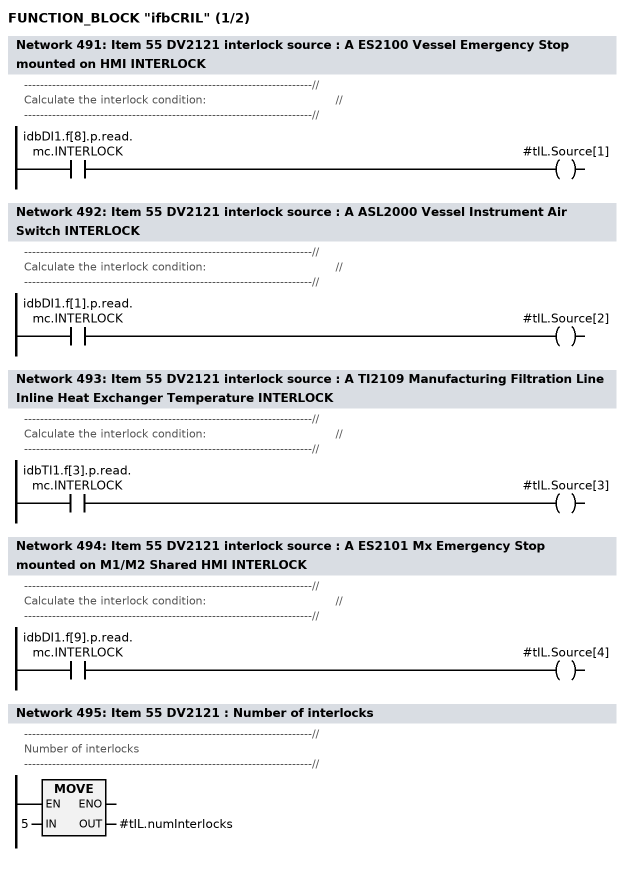
    A idbDI1.f[8].p.read.mc.INTERLOCK;
    = #tIL.Source[1];

NETWORK
TITLE = Item 55 DV2121 interlock source : A ASL2000 Vessel Instrument Air Switch INTERLOCK
    //------------------------------------------------------------------------//
    // Calculate the interlock condition:                                     //
    //------------------------------------------------------------------------//
    A idbDI1.f[1].p.read.mc.INTERLOCK;
    = #tIL.Source[2];

NETWORK
TITLE = Item 55 DV2121 interlock source : A TI2109 Manufacturing Filtration Line Inline Heat Exchanger Temperature INTERLOCK
    //------------------------------------------------------------------------//
    // Calculate the interlock condition:                                     //
    //------------------------------------------------------------------------//
    A idbTI1.f[3].p.read.mc.INTERLOCK;
    = #tIL.Source[3];

NETWORK
TITLE = Item 55 DV2121 interlock source : A ES2101 Mx Emergency Stop mounted on M1/M2 Shared HMI INTERLOCK
    //------------------------------------------------------------------------//
    // Calculate the interlock condition:                                     //
    //------------------------------------------------------------------------//
    A idbDI1.f[9].p.read.mc.INTERLOCK;
    = #tIL.Source[4];


NETWORK
TITLE = Item 55 DV2121 : Number of interlocks
    //------------------------------------------------------------------------//
    // Number of interlocks
    //------------------------------------------------------------------------//
    L 5;
    T #tIL.numInterlocks;

NETWORK
TITLE = Item 55 DV2121 : Aggregate individual interlocks into overall INTERLOCK flag
    //------------------------------------------------------------------------//
    // Determine if an interlock is raised:                                   //
    //------------------------------------------------------------------------//
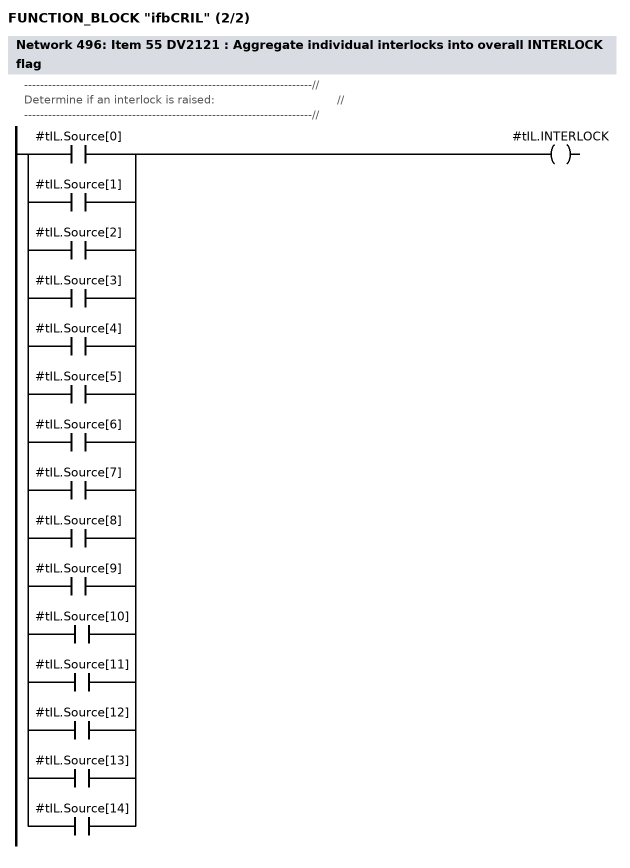
    O #tIL.Source[0];
    O #tIL.Source[1];
    O #tIL.Source[2];
    O #tIL.Source[3];
    O #tIL.Source[4];
    O #tIL.Source[5];
    O #tIL.Source[6];
    O #tIL.Source[7];
    O #tIL.Source[8];
    O #tIL.Source[9];
    O #tIL.Source[10];
    O #tIL.Source[11];
    O #tIL.Source[12];
    O #tIL.Source[13];
    O #tIL.Source[14];
    = #tIL.INTERLOCK;

NETWORK
TITLE = Item 55 DV2121 : Update the instance data
    //------------------------------------------------------------------------//
    // Update the instance DB with the calculated interlock flags:            //
    //------------------------------------------------------------------------//
    CALL MOVE
    {value_type := 'Variant'}
    (   IN                   := #tIL ,
        OUT                  := #p[55]
    );

NETWORK
TITLE = Item 56 DV2135 : SMFLx filter outlet drain valve initialise variables
    //------------------------------------------------------------------------//
    // CRITICAL INTERLOCK   CRITICAL INTERLOCK   CRITICAL INTERLOCK   CRITICA //
    // CRITICAL INTERLOCK   CRITICAL INTERLOCK   CRITICAL INTERLOCK   CRITICA //
    //                                                                        //
    // Clear the interlock flag:                                              //
    //------------------------------------------------------------------------//
    A "alwaysLow";
    = #tIL.INTERLOCK;

    //------------------------------------------------------------------------//
    // Clear all interlock values to initialise them to off:                  //
    //------------------------------------------------------------------------//
    CALL FILL_BLK
    {value_type := 'Bool', count_type := 'UInt'}
    (   IN                   := 0 ,
        COUNT                := 15 ,
        OUT                  := #tIL.Source[0]
    );


NETWORK
TITLE = Item 56 DV2135 interlock source : AN ZSC2111 MMFLx Filtration Inlet Flowpath Indicator IN   AN ZSC2109 SMFLx Filtration Line outlet Flowpath Indicator IN
    //------------------------------------------------------------------------//
    // Calculate the interlock condition:                                     //
    //------------------------------------------------------------------------//
    AN(;
    L "idbZSC2".f[11].p.read.mc.STATE;
    L "dbCONST".BLK.ZSC2.STATE.IN;
    ==I;
    );
AN(;
    L "idbZSC2".f[10].p.read.mc.STATE;
    L "dbCONST".BLK.ZSC2.STATE.IN;
    ==I;
    );
    = #tIL.Source[0];

NETWORK
TITLE = Item 56 DV2135 interlock source : A RD2101 Vessel Burst Disc ALARM
    //------------------------------------------------------------------------//
    // Calculate the interlock condition:                                     //
    //------------------------------------------------------------------------//
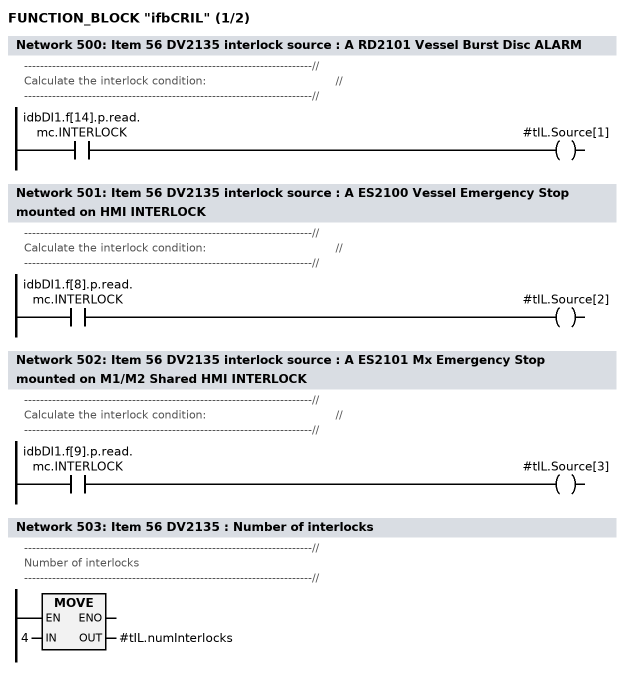
    A idbDI1.f[14].p.read.mc.INTERLOCK;
    = #tIL.Source[1];

NETWORK
TITLE = Item 56 DV2135 interlock source : A ES2100 Vessel Emergency Stop mounted on HMI INTERLOCK
    //------------------------------------------------------------------------//
    // Calculate the interlock condition:                                     //
    //------------------------------------------------------------------------//
    A idbDI1.f[8].p.read.mc.INTERLOCK;
    = #tIL.Source[2];

NETWORK
TITLE = Item 56 DV2135 interlock source : A ES2101 Mx Emergency Stop mounted on M1/M2 Shared HMI INTERLOCK
    //------------------------------------------------------------------------//
    // Calculate the interlock condition:                                     //
    //------------------------------------------------------------------------//
    A idbDI1.f[9].p.read.mc.INTERLOCK;
    = #tIL.Source[3];


NETWORK
TITLE = Item 56 DV2135 : Number of interlocks
    //------------------------------------------------------------------------//
    // Number of interlocks
    //------------------------------------------------------------------------//
    L 4;
    T #tIL.numInterlocks;

NETWORK
TITLE = Item 56 DV2135 : Aggregate individual interlocks into overall INTERLOCK flag
    //------------------------------------------------------------------------//
    // Determine if an interlock is raised:                                   //
    //------------------------------------------------------------------------//
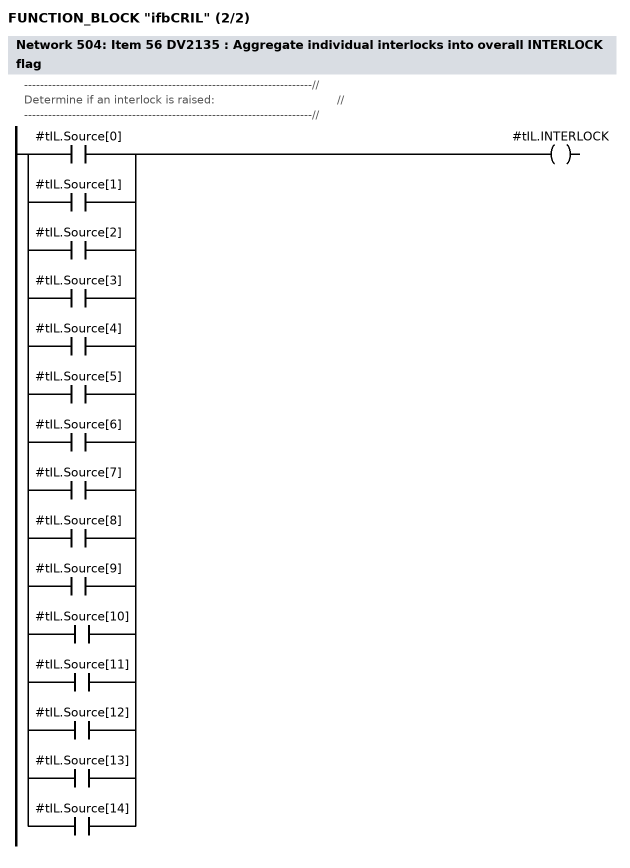
    O #tIL.Source[0];
    O #tIL.Source[1];
    O #tIL.Source[2];
    O #tIL.Source[3];
    O #tIL.Source[4];
    O #tIL.Source[5];
    O #tIL.Source[6];
    O #tIL.Source[7];
    O #tIL.Source[8];
    O #tIL.Source[9];
    O #tIL.Source[10];
    O #tIL.Source[11];
    O #tIL.Source[12];
    O #tIL.Source[13];
    O #tIL.Source[14];
    = #tIL.INTERLOCK;

NETWORK
TITLE = Item 56 DV2135 : Update the instance data
    //------------------------------------------------------------------------//
    // Update the instance DB with the calculated interlock flags:            //
    //------------------------------------------------------------------------//
    CALL MOVE
    {value_type := 'Variant'}
    (   IN                   := #tIL ,
        OUT                  := #p[56]
    );

NETWORK
TITLE = Item 57 DV2137 : SMFLx filter outlet valve initialise variables
    //------------------------------------------------------------------------//
    // CRITICAL INTERLOCK   CRITICAL INTERLOCK   CRITICAL INTERLOCK   CRITICA //
    // CRITICAL INTERLOCK   CRITICAL INTERLOCK   CRITICAL INTERLOCK   CRITICA //
    //                                                                        //
    // Clear the interlock flag:                                              //
    //------------------------------------------------------------------------//
    A "alwaysLow";
    = #tIL.INTERLOCK;

    //------------------------------------------------------------------------//
    // Clear all interlock values to initialise them to off:                  //
    //------------------------------------------------------------------------//
    CALL FILL_BLK
    {value_type := 'Bool', count_type := 'UInt'}
    (   IN                   := 0 ,
        COUNT                := 15 ,
        OUT                  := #tIL.Source[0]
    );


NETWORK
TITLE = Item 57 DV2137 interlock source : AN ZSC2111 MMFLx Filtration Inlet Flowpath Indicator IN   AN ZSC2109 SMFLx Filtration Line outlet Flowpath Indicator IN
    //------------------------------------------------------------------------//
    // Calculate the interlock condition:                                     //
    //------------------------------------------------------------------------//
    AN(;
    L "idbZSC2".f[11].p.read.mc.STATE;
    L "dbCONST".BLK.ZSC2.STATE.IN;
    ==I;
    );
AN(;
    L "idbZSC2".f[10].p.read.mc.STATE;
    L "dbCONST".BLK.ZSC2.STATE.IN;
    ==I;
    );
    = #tIL.Source[0];

NETWORK
TITLE = Item 57 DV2137 interlock source : A RD2101 Vessel Burst Disc ALARM
    //------------------------------------------------------------------------//
    // Calculate the interlock condition:                                     //
    //------------------------------------------------------------------------//
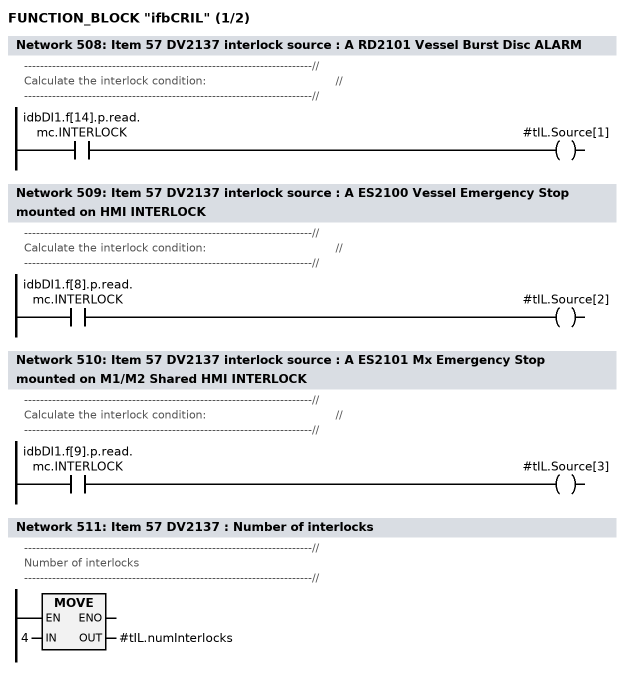
    A idbDI1.f[14].p.read.mc.INTERLOCK;
    = #tIL.Source[1];

NETWORK
TITLE = Item 57 DV2137 interlock source : A ES2100 Vessel Emergency Stop mounted on HMI INTERLOCK
    //------------------------------------------------------------------------//
    // Calculate the interlock condition:                                     //
    //------------------------------------------------------------------------//
    A idbDI1.f[8].p.read.mc.INTERLOCK;
    = #tIL.Source[2];

NETWORK
TITLE = Item 57 DV2137 interlock source : A ES2101 Mx Emergency Stop mounted on M1/M2 Shared HMI INTERLOCK
    //------------------------------------------------------------------------//
    // Calculate the interlock condition:                                     //
    //------------------------------------------------------------------------//
    A idbDI1.f[9].p.read.mc.INTERLOCK;
    = #tIL.Source[3];


NETWORK
TITLE = Item 57 DV2137 : Number of interlocks
    //------------------------------------------------------------------------//
    // Number of interlocks
    //------------------------------------------------------------------------//
    L 4;
    T #tIL.numInterlocks;

NETWORK
TITLE = Item 57 DV2137 : Aggregate individual interlocks into overall INTERLOCK flag
    //------------------------------------------------------------------------//
    // Determine if an interlock is raised:                                   //
    //------------------------------------------------------------------------//
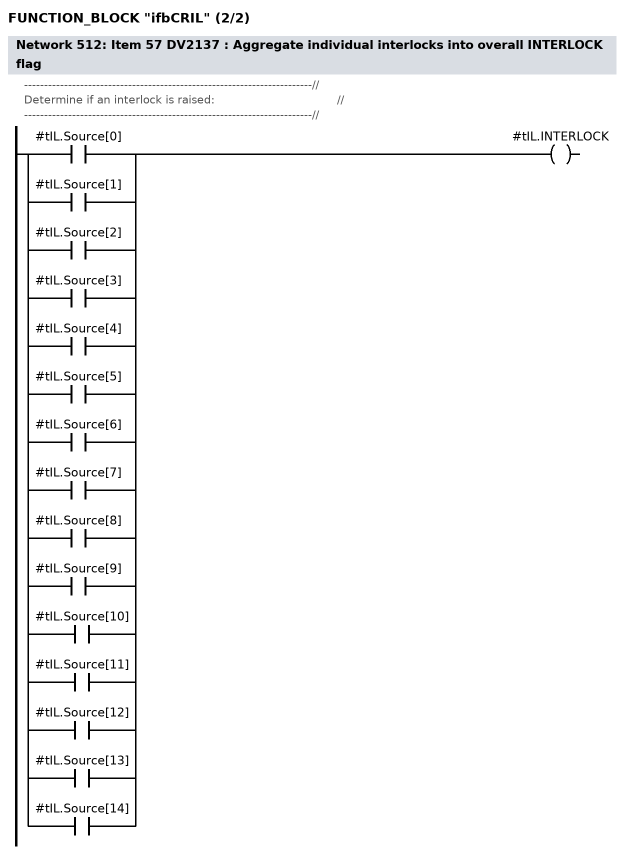
    O #tIL.Source[0];
    O #tIL.Source[1];
    O #tIL.Source[2];
    O #tIL.Source[3];
    O #tIL.Source[4];
    O #tIL.Source[5];
    O #tIL.Source[6];
    O #tIL.Source[7];
    O #tIL.Source[8];
    O #tIL.Source[9];
    O #tIL.Source[10];
    O #tIL.Source[11];
    O #tIL.Source[12];
    O #tIL.Source[13];
    O #tIL.Source[14];
    = #tIL.INTERLOCK;

NETWORK
TITLE = Item 57 DV2137 : Update the instance data
    //------------------------------------------------------------------------//
    // Update the instance DB with the calculated interlock flags:            //
    //------------------------------------------------------------------------//
    CALL MOVE
    {value_type := 'Variant'}
    (   IN                   := #tIL ,
        OUT                  := #p[57]
    );

NETWORK
TITLE = Item 58 DV2171 : MMFLx filter inlet drain valve initialise variables
    //------------------------------------------------------------------------//
    // CRITICAL INTERLOCK   CRITICAL INTERLOCK   CRITICAL INTERLOCK   CRITICA //
    // CRITICAL INTERLOCK   CRITICAL INTERLOCK   CRITICAL INTERLOCK   CRITICA //
    //                                                                        //
    // Clear the interlock flag:                                              //
    //------------------------------------------------------------------------//
    A "alwaysLow";
    = #tIL.INTERLOCK;

    //------------------------------------------------------------------------//
    // Clear all interlock values to initialise them to off:                  //
    //------------------------------------------------------------------------//
    CALL FILL_BLK
    {value_type := 'Bool', count_type := 'UInt'}
    (   IN                   := 0 ,
        COUNT                := 15 ,
        OUT                  := #tIL.Source[0]
    );


NETWORK
TITLE = Item 58 DV2171 interlock source : AN ZSC2113 MMFLx Filtration Inlet Flowpath Indicator IN   AN ZSC2115 MMFLx Filtration Inlet CIP & SIP Flowpath Indicator IN
    //------------------------------------------------------------------------//
    // Calculate the interlock condition:                                     //
    //------------------------------------------------------------------------//
    AN(;
    L "idbZSC2".f[12].p.read.mc.STATE;
    L "dbCONST".BLK.ZSC2.STATE.IN;
    ==I;
    );
AN(;
    L "idbZSC2".f[13].p.read.mc.STATE;
    L "dbCONST".BLK.ZSC2.STATE.IN;
    ==I;
    );
    = #tIL.Source[0];

NETWORK
TITLE = Item 58 DV2171 interlock source : AN ZSC2115 MMFLx Filtration Inlet CIP & SIP Flowpath Indicator IN
    //------------------------------------------------------------------------//
    // Calculate the interlock condition:                                     //
    //------------------------------------------------------------------------//
    AN(;
    L "idbZSC2".f[13].p.read.mc.STATE;
    L "dbCONST".BLK.ZSC2.STATE.IN;
    ==I;
    );
    = #tIL.Source[1];

NETWORK
TITLE = Item 58 DV2171 interlock source : A RD2101 Vessel Burst Disc ALARM
    //------------------------------------------------------------------------//
    // Calculate the interlock condition:                                     //
    //------------------------------------------------------------------------//
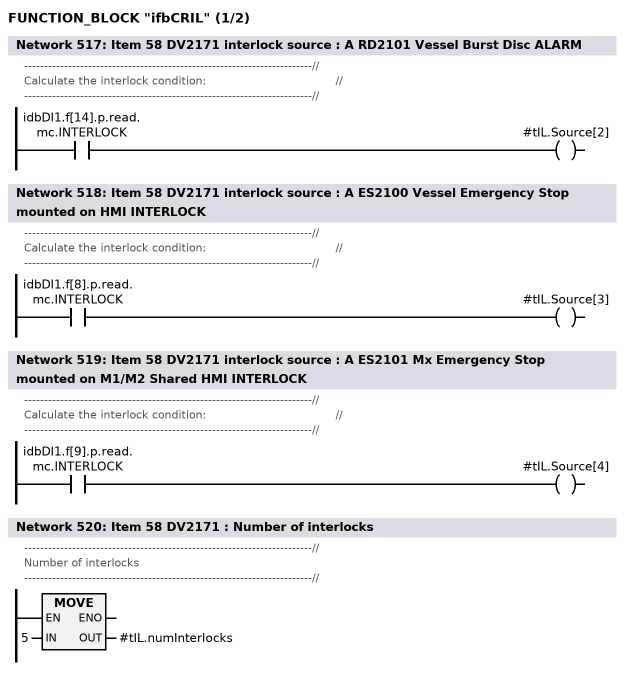
    A idbDI1.f[14].p.read.mc.INTERLOCK;
    = #tIL.Source[2];

NETWORK
TITLE = Item 58 DV2171 interlock source : A ES2100 Vessel Emergency Stop mounted on HMI INTERLOCK
    //------------------------------------------------------------------------//
    // Calculate the interlock condition:                                     //
    //------------------------------------------------------------------------//
    A idbDI1.f[8].p.read.mc.INTERLOCK;
    = #tIL.Source[3];

NETWORK
TITLE = Item 58 DV2171 interlock source : A ES2101 Mx Emergency Stop mounted on M1/M2 Shared HMI INTERLOCK
    //------------------------------------------------------------------------//
    // Calculate the interlock condition:                                     //
    //------------------------------------------------------------------------//
    A idbDI1.f[9].p.read.mc.INTERLOCK;
    = #tIL.Source[4];


NETWORK
TITLE = Item 58 DV2171 : Number of interlocks
    //------------------------------------------------------------------------//
    // Number of interlocks
    //------------------------------------------------------------------------//
    L 5;
    T #tIL.numInterlocks;

NETWORK
TITLE = Item 58 DV2171 : Aggregate individual interlocks into overall INTERLOCK flag
    //------------------------------------------------------------------------//
    // Determine if an interlock is raised:                                   //
    //------------------------------------------------------------------------//
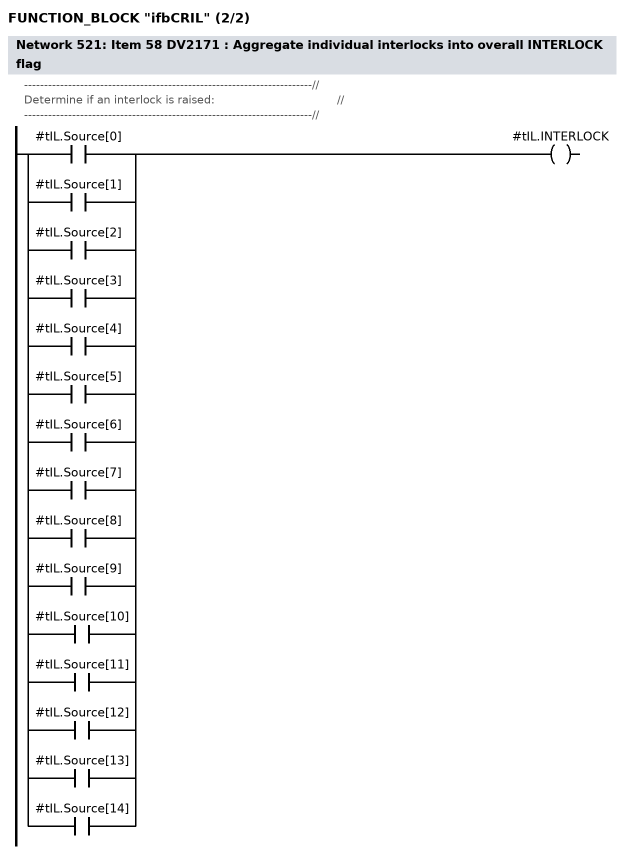
    O #tIL.Source[0];
    O #tIL.Source[1];
    O #tIL.Source[2];
    O #tIL.Source[3];
    O #tIL.Source[4];
    O #tIL.Source[5];
    O #tIL.Source[6];
    O #tIL.Source[7];
    O #tIL.Source[8];
    O #tIL.Source[9];
    O #tIL.Source[10];
    O #tIL.Source[11];
    O #tIL.Source[12];
    O #tIL.Source[13];
    O #tIL.Source[14];
    = #tIL.INTERLOCK;

NETWORK
TITLE = Item 58 DV2171 : Update the instance data
    //------------------------------------------------------------------------//
    // Update the instance DB with the calculated interlock flags:            //
    //------------------------------------------------------------------------//
    CALL MOVE
    {value_type := 'Variant'}
    (   IN                   := #tIL ,
        OUT                  := #p[58]
    );

NETWORK
TITLE = Item 59 DV2173 : MMFLx Inline Heat Exchanger inlet valve initialise variables
    //------------------------------------------------------------------------//
    // CRITICAL INTERLOCK   CRITICAL INTERLOCK   CRITICAL INTERLOCK   CRITICA //
    // CRITICAL INTERLOCK   CRITICAL INTERLOCK   CRITICAL INTERLOCK   CRITICA //
    //                                                                        //
    // Clear the interlock flag:                                              //
    //------------------------------------------------------------------------//
    A "alwaysLow";
    = #tIL.INTERLOCK;

    //------------------------------------------------------------------------//
    // Clear all interlock values to initialise them to off:                  //
    //------------------------------------------------------------------------//
    CALL FILL_BLK
    {value_type := 'Bool', count_type := 'UInt'}
    (   IN                   := 0 ,
        COUNT                := 15 ,
        OUT                  := #tIL.Source[0]
    );


NETWORK
TITLE = Item 59 DV2173 interlock source : AN ZSC2113 MMFLx Filtration Inlet Flowpath Indicator IN   AN ZSC2115 MMFLx Filtration Inlet CIP & SIP Flowpath Indicator IN
    //------------------------------------------------------------------------//
    // Calculate the interlock condition:                                     //
    //------------------------------------------------------------------------//
    AN(;
    L "idbZSC2".f[12].p.read.mc.STATE;
    L "dbCONST".BLK.ZSC2.STATE.IN;
    ==I;
    );
AN(;
    L "idbZSC2".f[13].p.read.mc.STATE;
    L "dbCONST".BLK.ZSC2.STATE.IN;
    ==I;
    );
    = #tIL.Source[0];

NETWORK
TITLE = Item 59 DV2173 interlock source : A RD2101 Vessel Burst Disc ALARM
    //------------------------------------------------------------------------//
    // Calculate the interlock condition:                                     //
    //------------------------------------------------------------------------//
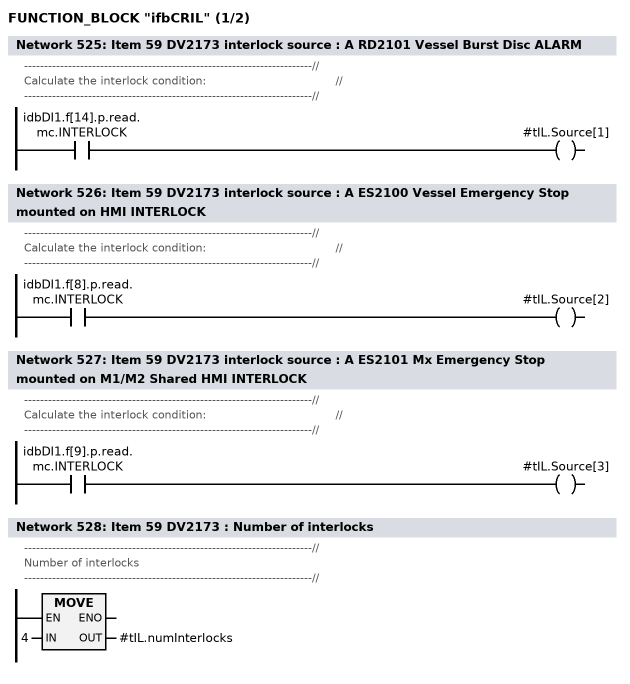
    A idbDI1.f[14].p.read.mc.INTERLOCK;
    = #tIL.Source[1];

NETWORK
TITLE = Item 59 DV2173 interlock source : A ES2100 Vessel Emergency Stop mounted on HMI INTERLOCK
    //------------------------------------------------------------------------//
    // Calculate the interlock condition:                                     //
    //------------------------------------------------------------------------//
    A idbDI1.f[8].p.read.mc.INTERLOCK;
    = #tIL.Source[2];

NETWORK
TITLE = Item 59 DV2173 interlock source : A ES2101 Mx Emergency Stop mounted on M1/M2 Shared HMI INTERLOCK
    //------------------------------------------------------------------------//
    // Calculate the interlock condition:                                     //
    //------------------------------------------------------------------------//
    A idbDI1.f[9].p.read.mc.INTERLOCK;
    = #tIL.Source[3];


NETWORK
TITLE = Item 59 DV2173 : Number of interlocks
    //------------------------------------------------------------------------//
    // Number of interlocks
    //------------------------------------------------------------------------//
    L 4;
    T #tIL.numInterlocks;

NETWORK
TITLE = Item 59 DV2173 : Aggregate individual interlocks into overall INTERLOCK flag
    //------------------------------------------------------------------------//
    // Determine if an interlock is raised:                                   //
    //------------------------------------------------------------------------//
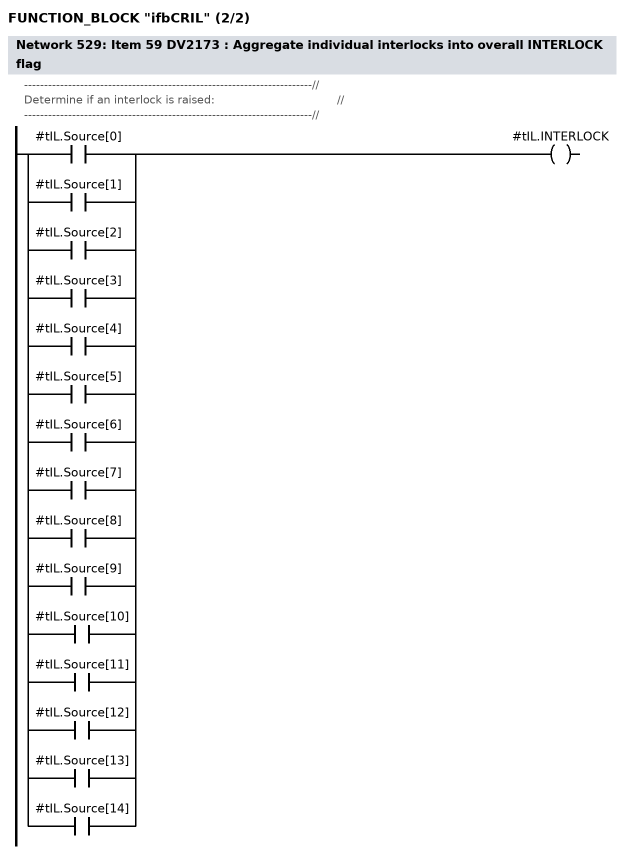
    O #tIL.Source[0];
    O #tIL.Source[1];
    O #tIL.Source[2];
    O #tIL.Source[3];
    O #tIL.Source[4];
    O #tIL.Source[5];
    O #tIL.Source[6];
    O #tIL.Source[7];
    O #tIL.Source[8];
    O #tIL.Source[9];
    O #tIL.Source[10];
    O #tIL.Source[11];
    O #tIL.Source[12];
    O #tIL.Source[13];
    O #tIL.Source[14];
    = #tIL.INTERLOCK;

NETWORK
TITLE = Item 59 DV2173 : Update the instance data
    //------------------------------------------------------------------------//
    // Update the instance DB with the calculated interlock flags:            //
    //------------------------------------------------------------------------//
    CALL MOVE
    {value_type := 'Variant'}
    (   IN                   := #tIL ,
        OUT                  := #p[59]
    );

NETWORK
TITLE = Item 60 DV3101 : Vent Valve initialise variables
    //------------------------------------------------------------------------//
    // CRITICAL INTERLOCK   CRITICAL INTERLOCK   CRITICAL INTERLOCK   CRITICA //
    // CRITICAL INTERLOCK   CRITICAL INTERLOCK   CRITICAL INTERLOCK   CRITICA //
    //                                                                        //
    // Clear the interlock flag:                                              //
    //------------------------------------------------------------------------//
    A "alwaysLow";
    = #tIL.INTERLOCK;

    //------------------------------------------------------------------------//
    // Clear all interlock values to initialise them to off:                  //
    //------------------------------------------------------------------------//
    CALL FILL_BLK
    {value_type := 'Bool', count_type := 'UInt'}
    (   IN                   := 0 ,
        COUNT                := 15 ,
        OUT                  := #tIL.Source[0]
    );


NETWORK
TITLE = Item 60 DV3101 interlock source : A RD3101 Vessel Burst Disc ALARM
    //------------------------------------------------------------------------//
    // Calculate the interlock condition:                                     //
    //------------------------------------------------------------------------//
    A idbDI1.f[15].p.read.mc.INTERLOCK;
    = #tIL.Source[0];

NETWORK
TITLE = Item 60 DV3101 interlock source : A ES3100 Vessel Emergency Stop mounted on HMI INTERLOCK
    //------------------------------------------------------------------------//
    // Calculate the interlock condition:                                     //
    //------------------------------------------------------------------------//
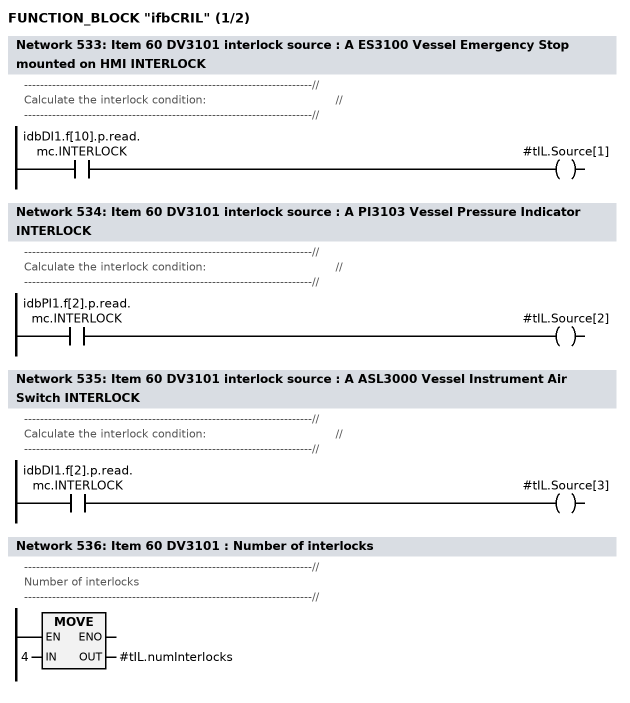
    A idbDI1.f[10].p.read.mc.INTERLOCK;
    = #tIL.Source[1];

NETWORK
TITLE = Item 60 DV3101 interlock source : A PI3103 Vessel Pressure Indicator INTERLOCK
    //------------------------------------------------------------------------//
    // Calculate the interlock condition:                                     //
    //------------------------------------------------------------------------//
    A idbPI1.f[2].p.read.mc.INTERLOCK;
    = #tIL.Source[2];

NETWORK
TITLE = Item 60 DV3101 interlock source : A ASL3000 Vessel Instrument Air Switch INTERLOCK
    //------------------------------------------------------------------------//
    // Calculate the interlock condition:                                     //
    //------------------------------------------------------------------------//
    A idbDI1.f[2].p.read.mc.INTERLOCK;
    = #tIL.Source[3];


NETWORK
TITLE = Item 60 DV3101 : Number of interlocks
    //------------------------------------------------------------------------//
    // Number of interlocks
    //------------------------------------------------------------------------//
    L 4;
    T #tIL.numInterlocks;

NETWORK
TITLE = Item 60 DV3101 : Aggregate individual interlocks into overall INTERLOCK flag
    //------------------------------------------------------------------------//
    // Determine if an interlock is raised:                                   //
    //------------------------------------------------------------------------//
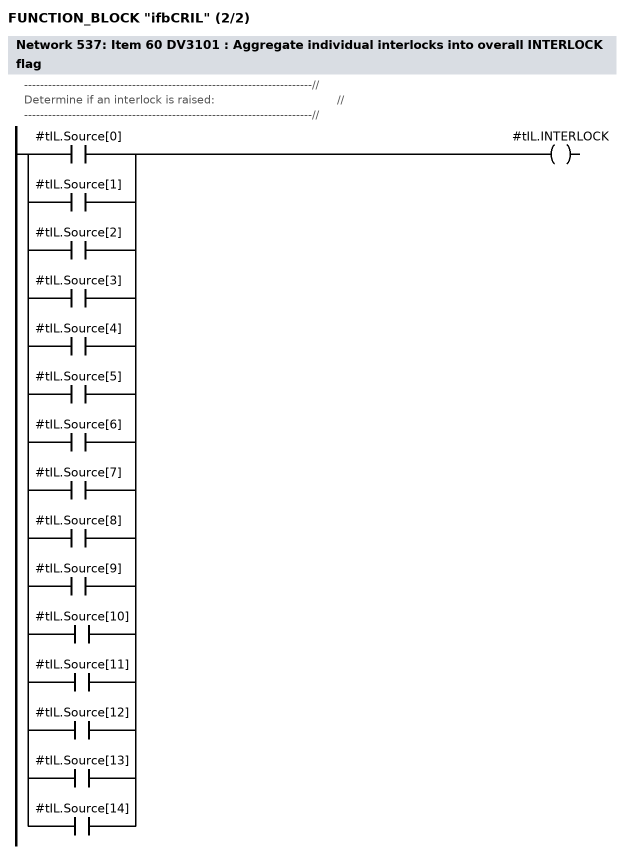
    O #tIL.Source[0];
    O #tIL.Source[1];
    O #tIL.Source[2];
    O #tIL.Source[3];
    O #tIL.Source[4];
    O #tIL.Source[5];
    O #tIL.Source[6];
    O #tIL.Source[7];
    O #tIL.Source[8];
    O #tIL.Source[9];
    O #tIL.Source[10];
    O #tIL.Source[11];
    O #tIL.Source[12];
    O #tIL.Source[13];
    O #tIL.Source[14];
    = #tIL.INTERLOCK;

NETWORK
TITLE = Item 60 DV3101 : Update the instance data
    //------------------------------------------------------------------------//
    // Update the instance DB with the calculated interlock flags:            //
    //------------------------------------------------------------------------//
    CALL MOVE
    {value_type := 'Variant'}
    (   IN                   := #tIL ,
        OUT                  := #p[60]
    );

NETWORK
TITLE = Item 61 DV3103 : HP CA Supply Valve initialise variables
    //------------------------------------------------------------------------//
    // CRITICAL INTERLOCK   CRITICAL INTERLOCK   CRITICAL INTERLOCK   CRITICA //
    // CRITICAL INTERLOCK   CRITICAL INTERLOCK   CRITICAL INTERLOCK   CRITICA //
    //                                                                        //
    // Clear the interlock flag:                                              //
    //------------------------------------------------------------------------//
    A "alwaysLow";
    = #tIL.INTERLOCK;

    //------------------------------------------------------------------------//
    // Clear all interlock values to initialise them to off:                  //
    //------------------------------------------------------------------------//
    CALL FILL_BLK
    {value_type := 'Bool', count_type := 'UInt'}
    (   IN                   := 0 ,
        COUNT                := 15 ,
        OUT                  := #tIL.Source[0]
    );


NETWORK
TITLE = Item 61 DV3103 interlock source : A RD3101 Vessel Burst Disc ALARM
    //------------------------------------------------------------------------//
    // Calculate the interlock condition:                                     //
    //------------------------------------------------------------------------//
    A idbDI1.f[15].p.read.mc.INTERLOCK;
    = #tIL.Source[0];

NETWORK
TITLE = Item 61 DV3103 interlock source : A ES3100 Vessel Emergency Stop mounted on HMI INTERLOCK
    //------------------------------------------------------------------------//
    // Calculate the interlock condition:                                     //
    //------------------------------------------------------------------------//
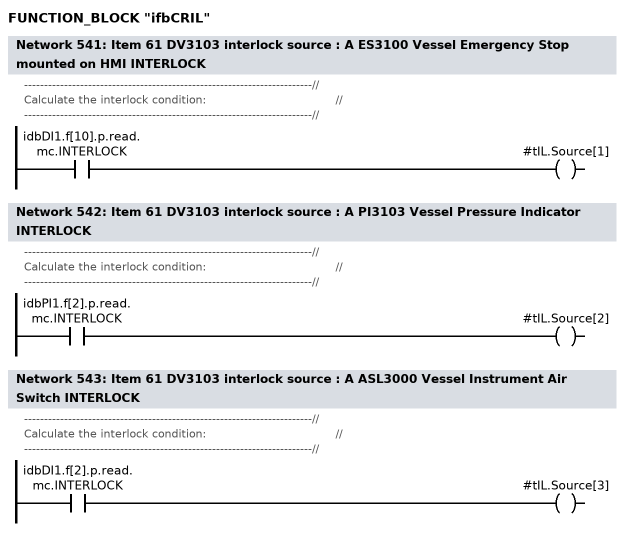
    A idbDI1.f[10].p.read.mc.INTERLOCK;
    = #tIL.Source[1];

NETWORK
TITLE = Item 61 DV3103 interlock source : A PI3103 Vessel Pressure Indicator INTERLOCK
    //------------------------------------------------------------------------//
    // Calculate the interlock condition:                                     //
    //------------------------------------------------------------------------//
    A idbPI1.f[2].p.read.mc.INTERLOCK;
    = #tIL.Source[2];

NETWORK
TITLE = Item 61 DV3103 interlock source : A ASL3000 Vessel Instrument Air Switch INTERLOCK
    //------------------------------------------------------------------------//
    // Calculate the interlock condition:                                     //
    //------------------------------------------------------------------------//
    A idbDI1.f[2].p.read.mc.INTERLOCK;
    = #tIL.Source[3];

NETWORK
TITLE = Item 61 DV3103 interlock source : AN ZSC3101 Vessel Manway Closed Indicator CLOSED
    //------------------------------------------------------------------------//
    // Calculate the interlock condition:                                     //
    //------------------------------------------------------------------------//
    AN(;
    L "idbZSC1".f[2].p.read.mc.STATE;
    L "dbCONST".BLK.ZSC1.STATE.CLOSED;
    ==I;
    );
    = #tIL.Source[4];


NETWORK
TITLE = Item 61 DV3103 : Number of interlocks
    //------------------------------------------------------------------------//
    // Number of interlocks
    //------------------------------------------------------------------------//
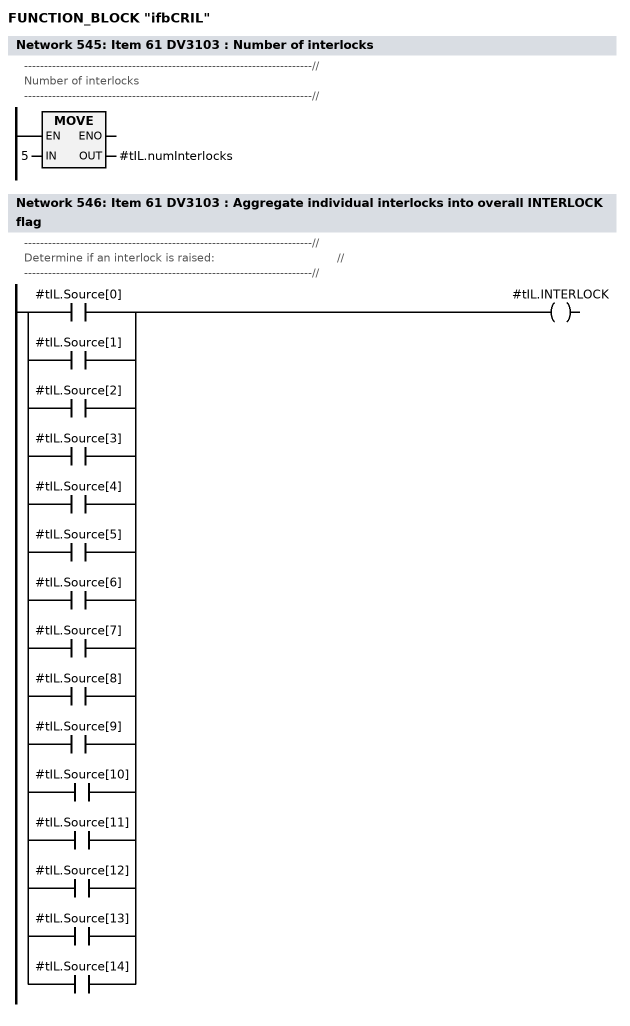
    L 5;
    T #tIL.numInterlocks;

NETWORK
TITLE = Item 61 DV3103 : Aggregate individual interlocks into overall INTERLOCK flag
    //------------------------------------------------------------------------//
    // Determine if an interlock is raised:                                   //
    //------------------------------------------------------------------------//
    O #tIL.Source[0];
    O #tIL.Source[1];
    O #tIL.Source[2];
    O #tIL.Source[3];
    O #tIL.Source[4];
    O #tIL.Source[5];
    O #tIL.Source[6];
    O #tIL.Source[7];
    O #tIL.Source[8];
    O #tIL.Source[9];
    O #tIL.Source[10];
    O #tIL.Source[11];
    O #tIL.Source[12];
    O #tIL.Source[13];
    O #tIL.Source[14];
    = #tIL.INTERLOCK;

NETWORK
TITLE = Item 61 DV3103 : Update the instance data
    //------------------------------------------------------------------------//
    // Update the instance DB with the calculated interlock flags:            //
    //------------------------------------------------------------------------//
    CALL MOVE
    {value_type := 'Variant'}
    (   IN                   := #tIL ,
        OUT                  := #p[61]
    );

NETWORK
TITLE = Item 62 DV3105 : LP CA Supply Valve initialise variables
    //------------------------------------------------------------------------//
    // CRITICAL INTERLOCK   CRITICAL INTERLOCK   CRITICAL INTERLOCK   CRITICA //
    // CRITICAL INTERLOCK   CRITICAL INTERLOCK   CRITICAL INTERLOCK   CRITICA //
    //                                                                        //
    // Clear the interlock flag:                                              //
    //------------------------------------------------------------------------//
    A "alwaysLow";
    = #tIL.INTERLOCK;

    //------------------------------------------------------------------------//
    // Clear all interlock values to initialise them to off:                  //
    //------------------------------------------------------------------------//
    CALL FILL_BLK
    {value_type := 'Bool', count_type := 'UInt'}
    (   IN                   := 0 ,
        COUNT                := 15 ,
        OUT                  := #tIL.Source[0]
    );


NETWORK
TITLE = Item 62 DV3105 interlock source : A RD3101 Vessel Burst Disc ALARM
    //------------------------------------------------------------------------//
    // Calculate the interlock condition:                                     //
    //------------------------------------------------------------------------//
    A idbDI1.f[15].p.read.mc.INTERLOCK;
    = #tIL.Source[0];

NETWORK
TITLE = Item 62 DV3105 interlock source : A ES3100 Vessel Emergency Stop mounted on HMI INTERLOCK
    //------------------------------------------------------------------------//
    // Calculate the interlock condition:                                     //
    //------------------------------------------------------------------------//
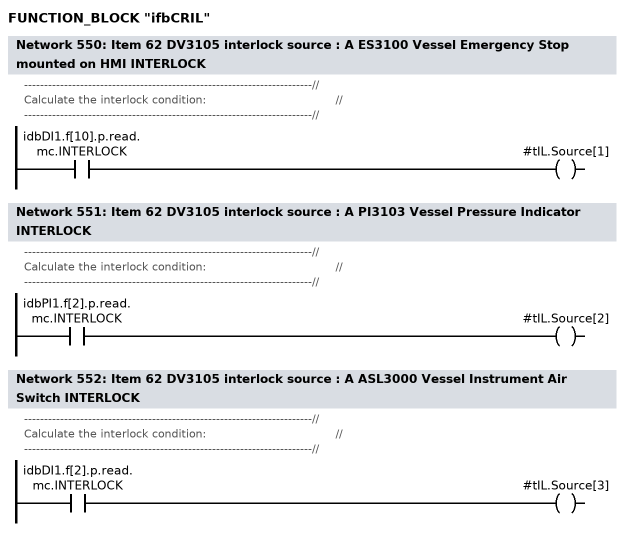
    A idbDI1.f[10].p.read.mc.INTERLOCK;
    = #tIL.Source[1];

NETWORK
TITLE = Item 62 DV3105 interlock source : A PI3103 Vessel Pressure Indicator INTERLOCK
    //------------------------------------------------------------------------//
    // Calculate the interlock condition:                                     //
    //------------------------------------------------------------------------//
    A idbPI1.f[2].p.read.mc.INTERLOCK;
    = #tIL.Source[2];

NETWORK
TITLE = Item 62 DV3105 interlock source : A ASL3000 Vessel Instrument Air Switch INTERLOCK
    //------------------------------------------------------------------------//
    // Calculate the interlock condition:                                     //
    //------------------------------------------------------------------------//
    A idbDI1.f[2].p.read.mc.INTERLOCK;
    = #tIL.Source[3];

NETWORK
TITLE = Item 62 DV3105 interlock source : AN ZSC3101 Vessel Manway Closed Indicator CLOSED
    //------------------------------------------------------------------------//
    // Calculate the interlock condition:                                     //
    //------------------------------------------------------------------------//
    AN(;
    L "idbZSC1".f[2].p.read.mc.STATE;
    L "dbCONST".BLK.ZSC1.STATE.CLOSED;
    ==I;
    );
    = #tIL.Source[4];


NETWORK
TITLE = Item 62 DV3105 : Number of interlocks
    //------------------------------------------------------------------------//
    // Number of interlocks
    //------------------------------------------------------------------------//
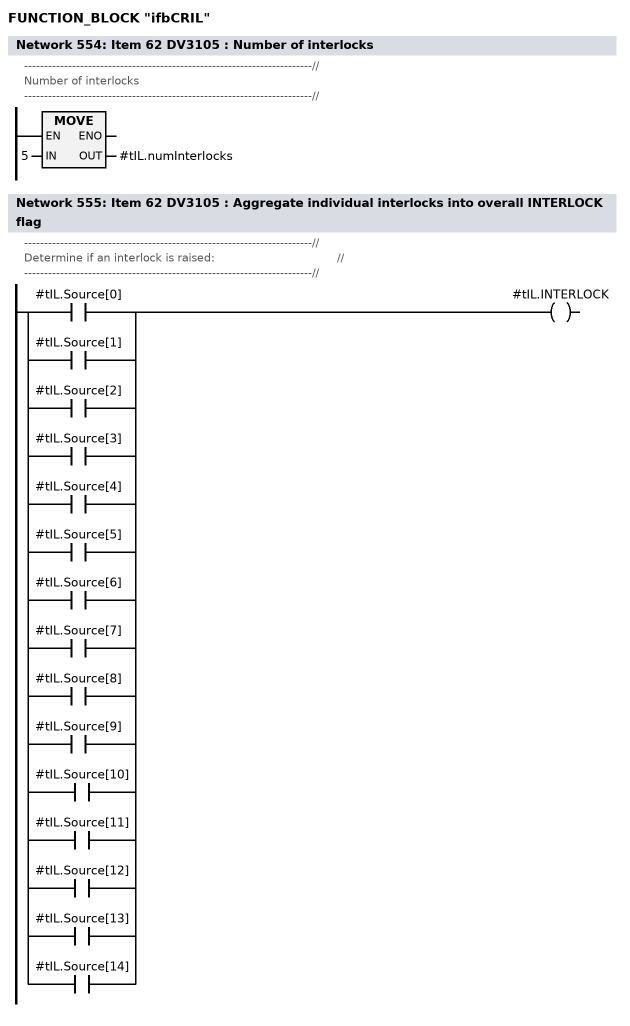
    L 5;
    T #tIL.numInterlocks;

NETWORK
TITLE = Item 62 DV3105 : Aggregate individual interlocks into overall INTERLOCK flag
    //------------------------------------------------------------------------//
    // Determine if an interlock is raised:                                   //
    //------------------------------------------------------------------------//
    O #tIL.Source[0];
    O #tIL.Source[1];
    O #tIL.Source[2];
    O #tIL.Source[3];
    O #tIL.Source[4];
    O #tIL.Source[5];
    O #tIL.Source[6];
    O #tIL.Source[7];
    O #tIL.Source[8];
    O #tIL.Source[9];
    O #tIL.Source[10];
    O #tIL.Source[11];
    O #tIL.Source[12];
    O #tIL.Source[13];
    O #tIL.Source[14];
    = #tIL.INTERLOCK;

NETWORK
TITLE = Item 62 DV3105 : Update the instance data
    //------------------------------------------------------------------------//
    // Update the instance DB with the calculated interlock flags:            //
    //------------------------------------------------------------------------//
    CALL MOVE
    {value_type := 'Variant'}
    (   IN                   := #tIL ,
        OUT                  := #p[62]
    );

NETWORK
TITLE = Item 63 DV3107 : Vacuum valve initialise variables
    //------------------------------------------------------------------------//
    // CRITICAL INTERLOCK   CRITICAL INTERLOCK   CRITICAL INTERLOCK   CRITICA //
    // CRITICAL INTERLOCK   CRITICAL INTERLOCK   CRITICAL INTERLOCK   CRITICA //
    //                                                                        //
    // Clear the interlock flag:                                              //
    //------------------------------------------------------------------------//
    A "alwaysLow";
    = #tIL.INTERLOCK;

    //------------------------------------------------------------------------//
    // Clear all interlock values to initialise them to off:                  //
    //------------------------------------------------------------------------//
    CALL FILL_BLK
    {value_type := 'Bool', count_type := 'UInt'}
    (   IN                   := 0 ,
        COUNT                := 15 ,
        OUT                  := #tIL.Source[0]
    );


NETWORK
TITLE = Item 63 DV3107 interlock source : A RD3101 Vessel Burst Disc ALARM
    //------------------------------------------------------------------------//
    // Calculate the interlock condition:                                     //
    //------------------------------------------------------------------------//
    A idbDI1.f[15].p.read.mc.INTERLOCK;
    = #tIL.Source[0];

NETWORK
TITLE = Item 63 DV3107 interlock source : A ES3100 Vessel Emergency Stop mounted on HMI INTERLOCK
    //------------------------------------------------------------------------//
    // Calculate the interlock condition:                                     //
    //------------------------------------------------------------------------//
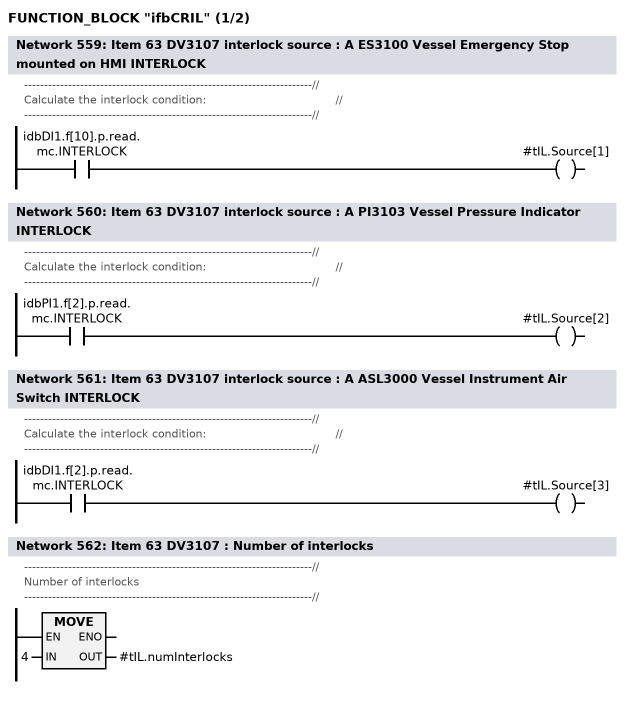
    A idbDI1.f[10].p.read.mc.INTERLOCK;
    = #tIL.Source[1];

NETWORK
TITLE = Item 63 DV3107 interlock source : A PI3103 Vessel Pressure Indicator INTERLOCK
    //------------------------------------------------------------------------//
    // Calculate the interlock condition:                                     //
    //------------------------------------------------------------------------//
    A idbPI1.f[2].p.read.mc.INTERLOCK;
    = #tIL.Source[2];

NETWORK
TITLE = Item 63 DV3107 interlock source : A ASL3000 Vessel Instrument Air Switch INTERLOCK
    //------------------------------------------------------------------------//
    // Calculate the interlock condition:                                     //
    //------------------------------------------------------------------------//
    A idbDI1.f[2].p.read.mc.INTERLOCK;
    = #tIL.Source[3];


NETWORK
TITLE = Item 63 DV3107 : Number of interlocks
    //------------------------------------------------------------------------//
    // Number of interlocks
    //------------------------------------------------------------------------//
    L 4;
    T #tIL.numInterlocks;

NETWORK
TITLE = Item 63 DV3107 : Aggregate individual interlocks into overall INTERLOCK flag
    //------------------------------------------------------------------------//
    // Determine if an interlock is raised:                                   //
    //------------------------------------------------------------------------//
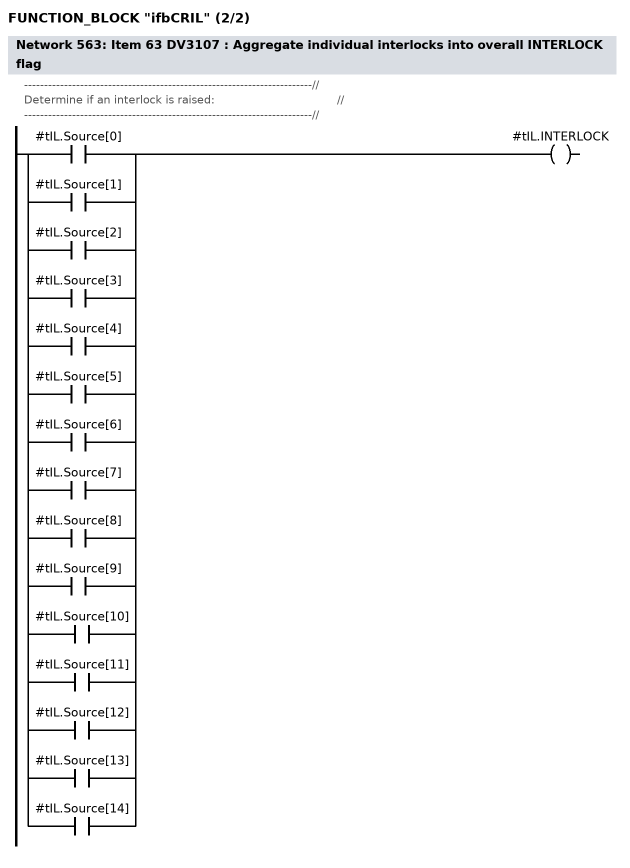
    O #tIL.Source[0];
    O #tIL.Source[1];
    O #tIL.Source[2];
    O #tIL.Source[3];
    O #tIL.Source[4];
    O #tIL.Source[5];
    O #tIL.Source[6];
    O #tIL.Source[7];
    O #tIL.Source[8];
    O #tIL.Source[9];
    O #tIL.Source[10];
    O #tIL.Source[11];
    O #tIL.Source[12];
    O #tIL.Source[13];
    O #tIL.Source[14];
    = #tIL.INTERLOCK;

NETWORK
TITLE = Item 63 DV3107 : Update the instance data
    //------------------------------------------------------------------------//
    // Update the instance DB with the calculated interlock flags:            //
    //------------------------------------------------------------------------//
    CALL MOVE
    {value_type := 'Variant'}
    (   IN                   := #tIL ,
        OUT                  := #p[63]
    );

NETWORK
TITLE = Item 64 DV3109 : PS Supply for WFI Loop initialise variables
    //------------------------------------------------------------------------//
    // CRITICAL INTERLOCK   CRITICAL INTERLOCK   CRITICAL INTERLOCK   CRITICA //
    // CRITICAL INTERLOCK   CRITICAL INTERLOCK   CRITICAL INTERLOCK   CRITICA //
    //                                                                        //
    // Clear the interlock flag:                                              //
    //------------------------------------------------------------------------//
    A "alwaysLow";
    = #tIL.INTERLOCK;

    //------------------------------------------------------------------------//
    // Clear all interlock values to initialise them to off:                  //
    //------------------------------------------------------------------------//
    CALL FILL_BLK
    {value_type := 'Bool', count_type := 'UInt'}
    (   IN                   := 0 ,
        COUNT                := 15 ,
        OUT                  := #tIL.Source[0]
    );


NETWORK
TITLE = Item 64 DV3109 interlock source : ON ZSC3107 Vessel inlet line Flowpath Indicator IN   ON ZSC3103 Vessel WFI Supply Flowpath Indicator IN
    //------------------------------------------------------------------------//
    // Calculate the interlock condition:                                     //
    //------------------------------------------------------------------------//
    ON(;
    L "idbZSC2".f[16].p.read.mc.STATE;
    L "dbCONST".BLK.ZSC2.STATE.IN;
    ==I;
    );
ON(;
    L "idbZSC2".f[14].p.read.mc.STATE;
    L "dbCONST".BLK.ZSC2.STATE.IN;
    ==I;
    );
    = #tIL.Source[0];

NETWORK
TITLE = Item 64 DV3109 interlock source : A DV3111 Vessel WFI Supply Valve OPENED
    //------------------------------------------------------------------------//
    // Calculate the interlock condition:                                     //
    //------------------------------------------------------------------------//
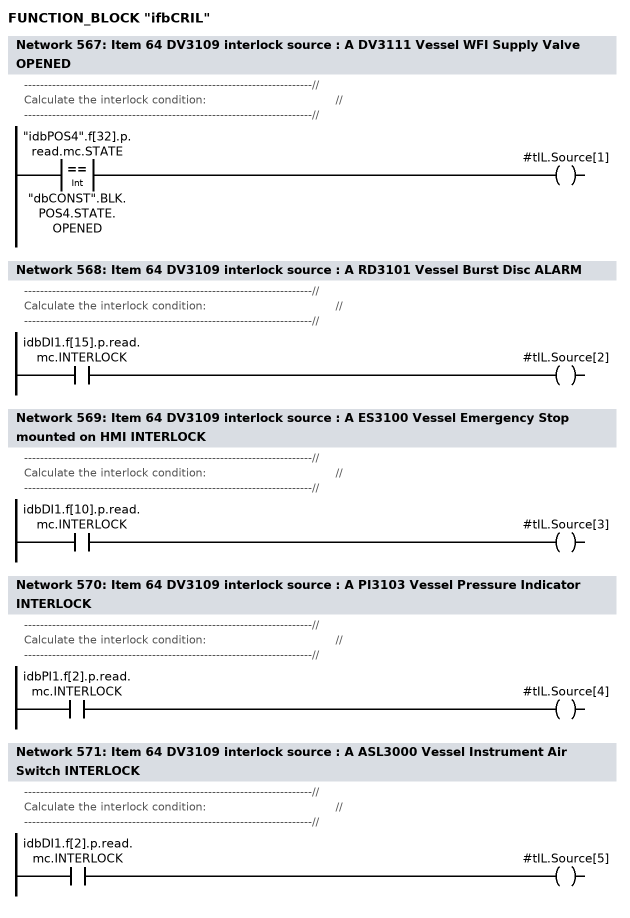
    A(;
    L "idbPOS4".f[32].p.read.mc.STATE;
    L "dbCONST".BLK.POS4.STATE.OPENED;
    ==I;
    );
    = #tIL.Source[1];

NETWORK
TITLE = Item 64 DV3109 interlock source : A RD3101 Vessel Burst Disc ALARM
    //------------------------------------------------------------------------//
    // Calculate the interlock condition:                                     //
    //------------------------------------------------------------------------//
    A idbDI1.f[15].p.read.mc.INTERLOCK;
    = #tIL.Source[2];

NETWORK
TITLE = Item 64 DV3109 interlock source : A ES3100 Vessel Emergency Stop mounted on HMI INTERLOCK
    //------------------------------------------------------------------------//
    // Calculate the interlock condition:                                     //
    //------------------------------------------------------------------------//
    A idbDI1.f[10].p.read.mc.INTERLOCK;
    = #tIL.Source[3];

NETWORK
TITLE = Item 64 DV3109 interlock source : A PI3103 Vessel Pressure Indicator INTERLOCK
    //------------------------------------------------------------------------//
    // Calculate the interlock condition:                                     //
    //------------------------------------------------------------------------//
    A idbPI1.f[2].p.read.mc.INTERLOCK;
    = #tIL.Source[4];

NETWORK
TITLE = Item 64 DV3109 interlock source : A ASL3000 Vessel Instrument Air Switch INTERLOCK
    //------------------------------------------------------------------------//
    // Calculate the interlock condition:                                     //
    //------------------------------------------------------------------------//
    A idbDI1.f[2].p.read.mc.INTERLOCK;
    = #tIL.Source[5];

NETWORK
TITLE = Item 64 DV3109 interlock source : AN ZSC3101 Vessel Manway Closed Indicator CLOSED
    //------------------------------------------------------------------------//
    // Calculate the interlock condition:                                     //
    //------------------------------------------------------------------------//
    AN(;
    L "idbZSC1".f[2].p.read.mc.STATE;
    L "dbCONST".BLK.ZSC1.STATE.CLOSED;
    ==I;
    );
    = #tIL.Source[6];


NETWORK
TITLE = Item 64 DV3109 : Number of interlocks
    //------------------------------------------------------------------------//
    // Number of interlocks
    //------------------------------------------------------------------------//
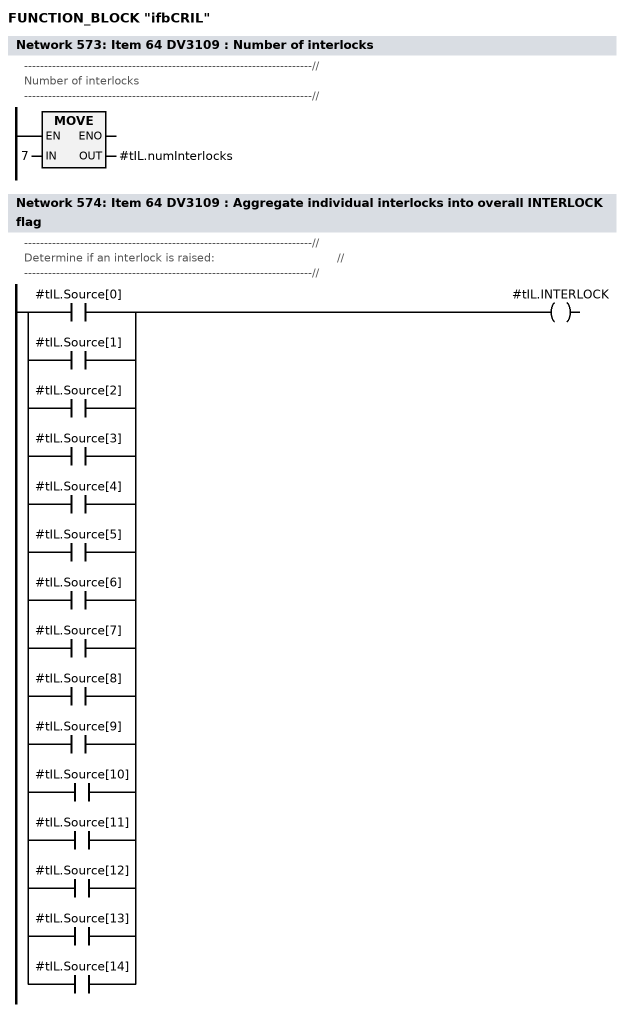
    L 7;
    T #tIL.numInterlocks;

NETWORK
TITLE = Item 64 DV3109 : Aggregate individual interlocks into overall INTERLOCK flag
    //------------------------------------------------------------------------//
    // Determine if an interlock is raised:                                   //
    //------------------------------------------------------------------------//
    O #tIL.Source[0];
    O #tIL.Source[1];
    O #tIL.Source[2];
    O #tIL.Source[3];
    O #tIL.Source[4];
    O #tIL.Source[5];
    O #tIL.Source[6];
    O #tIL.Source[7];
    O #tIL.Source[8];
    O #tIL.Source[9];
    O #tIL.Source[10];
    O #tIL.Source[11];
    O #tIL.Source[12];
    O #tIL.Source[13];
    O #tIL.Source[14];
    = #tIL.INTERLOCK;

NETWORK
TITLE = Item 64 DV3109 : Update the instance data
    //------------------------------------------------------------------------//
    // Update the instance DB with the calculated interlock flags:            //
    //------------------------------------------------------------------------//
    CALL MOVE
    {value_type := 'Variant'}
    (   IN                   := #tIL ,
        OUT                  := #p[64]
    );

NETWORK
TITLE = Item 65 DV3111 : WFI Supply Valve initialise variables
    //------------------------------------------------------------------------//
    // CRITICAL INTERLOCK   CRITICAL INTERLOCK   CRITICAL INTERLOCK   CRITICA //
    // CRITICAL INTERLOCK   CRITICAL INTERLOCK   CRITICAL INTERLOCK   CRITICA //
    //                                                                        //
    // Clear the interlock flag:                                              //
    //------------------------------------------------------------------------//
    A "alwaysLow";
    = #tIL.INTERLOCK;

    //------------------------------------------------------------------------//
    // Clear all interlock values to initialise them to off:                  //
    //------------------------------------------------------------------------//
    CALL FILL_BLK
    {value_type := 'Bool', count_type := 'UInt'}
    (   IN                   := 0 ,
        COUNT                := 15 ,
        OUT                  := #tIL.Source[0]
    );


NETWORK
TITLE = Item 65 DV3111 interlock source : ON ZSC3107 Vessel inlet line Flowpath Indicator IN   ON ZSC3103 Vessel WFI Supply Flowpath Indicator IN
    //------------------------------------------------------------------------//
    // Calculate the interlock condition:                                     //
    //------------------------------------------------------------------------//
    ON(;
    L "idbZSC2".f[16].p.read.mc.STATE;
    L "dbCONST".BLK.ZSC2.STATE.IN;
    ==I;
    );
ON(;
    L "idbZSC2".f[14].p.read.mc.STATE;
    L "dbCONST".BLK.ZSC2.STATE.IN;
    ==I;
    );
    = #tIL.Source[0];

NETWORK
TITLE = Item 65 DV3111 interlock source : A DV3109 Vessel PS Supply for WFI Loop OPENED
    //------------------------------------------------------------------------//
    // Calculate the interlock condition:                                     //
    //------------------------------------------------------------------------//
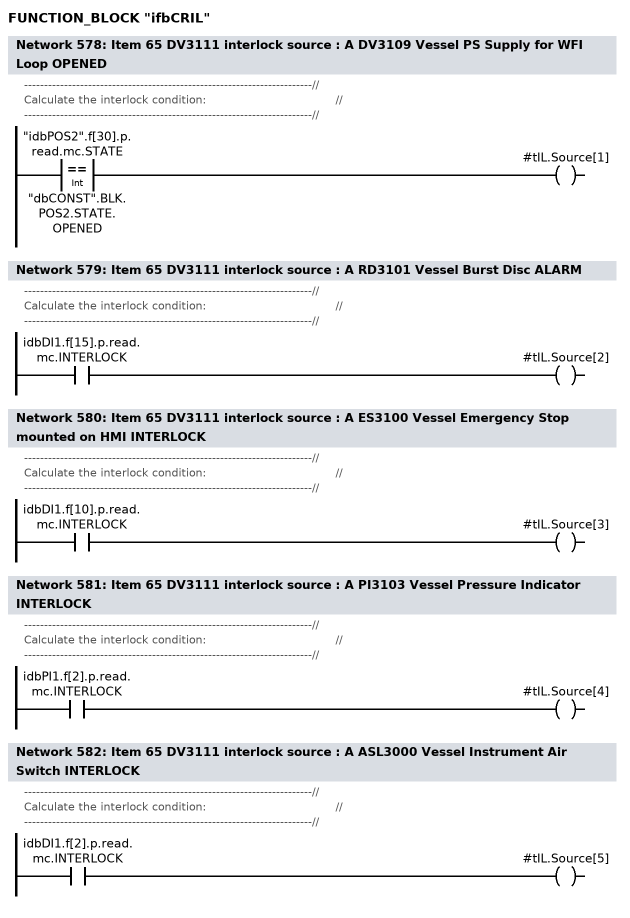
    A(;
    L "idbPOS2".f[30].p.read.mc.STATE;
    L "dbCONST".BLK.POS2.STATE.OPENED;
    ==I;
    );
    = #tIL.Source[1];

NETWORK
TITLE = Item 65 DV3111 interlock source : A RD3101 Vessel Burst Disc ALARM
    //------------------------------------------------------------------------//
    // Calculate the interlock condition:                                     //
    //------------------------------------------------------------------------//
    A idbDI1.f[15].p.read.mc.INTERLOCK;
    = #tIL.Source[2];

NETWORK
TITLE = Item 65 DV3111 interlock source : A ES3100 Vessel Emergency Stop mounted on HMI INTERLOCK
    //------------------------------------------------------------------------//
    // Calculate the interlock condition:                                     //
    //------------------------------------------------------------------------//
    A idbDI1.f[10].p.read.mc.INTERLOCK;
    = #tIL.Source[3];

NETWORK
TITLE = Item 65 DV3111 interlock source : A PI3103 Vessel Pressure Indicator INTERLOCK
    //------------------------------------------------------------------------//
    // Calculate the interlock condition:                                     //
    //------------------------------------------------------------------------//
    A idbPI1.f[2].p.read.mc.INTERLOCK;
    = #tIL.Source[4];

NETWORK
TITLE = Item 65 DV3111 interlock source : A ASL3000 Vessel Instrument Air Switch INTERLOCK
    //------------------------------------------------------------------------//
    // Calculate the interlock condition:                                     //
    //------------------------------------------------------------------------//
    A idbDI1.f[2].p.read.mc.INTERLOCK;
    = #tIL.Source[5];

NETWORK
TITLE = Item 65 DV3111 interlock source : AN ZSC3101 Vessel Manway Closed Indicator CLOSED
    //------------------------------------------------------------------------//
    // Calculate the interlock condition:                                     //
    //------------------------------------------------------------------------//
    AN(;
    L "idbZSC1".f[2].p.read.mc.STATE;
    L "dbCONST".BLK.ZSC1.STATE.CLOSED;
    ==I;
    );
    = #tIL.Source[6];


NETWORK
TITLE = Item 65 DV3111 : Number of interlocks
    //------------------------------------------------------------------------//
    // Number of interlocks
    //------------------------------------------------------------------------//
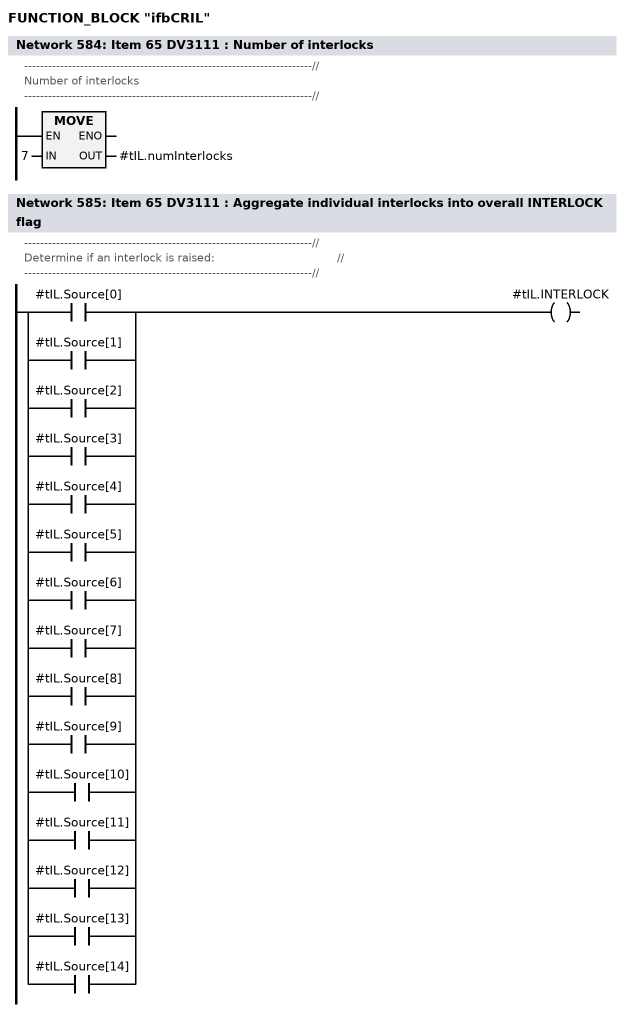
    L 7;
    T #tIL.numInterlocks;

NETWORK
TITLE = Item 65 DV3111 : Aggregate individual interlocks into overall INTERLOCK flag
    //------------------------------------------------------------------------//
    // Determine if an interlock is raised:                                   //
    //------------------------------------------------------------------------//
    O #tIL.Source[0];
    O #tIL.Source[1];
    O #tIL.Source[2];
    O #tIL.Source[3];
    O #tIL.Source[4];
    O #tIL.Source[5];
    O #tIL.Source[6];
    O #tIL.Source[7];
    O #tIL.Source[8];
    O #tIL.Source[9];
    O #tIL.Source[10];
    O #tIL.Source[11];
    O #tIL.Source[12];
    O #tIL.Source[13];
    O #tIL.Source[14];
    = #tIL.INTERLOCK;

NETWORK
TITLE = Item 65 DV3111 : Update the instance data
    //------------------------------------------------------------------------//
    // Update the instance DB with the calculated interlock flags:            //
    //------------------------------------------------------------------------//
    CALL MOVE
    {value_type := 'Variant'}
    (   IN                   := #tIL ,
        OUT                  := #p[65]
    );

NETWORK
TITLE = Item 66 DV3113 : PW Supply Valve initialise variables
    //------------------------------------------------------------------------//
    // CRITICAL INTERLOCK   CRITICAL INTERLOCK   CRITICAL INTERLOCK   CRITICA //
    // CRITICAL INTERLOCK   CRITICAL INTERLOCK   CRITICAL INTERLOCK   CRITICA //
    //                                                                        //
    // Clear the interlock flag:                                              //
    //------------------------------------------------------------------------//
    A "alwaysLow";
    = #tIL.INTERLOCK;

    //------------------------------------------------------------------------//
    // Clear all interlock values to initialise them to off:                  //
    //------------------------------------------------------------------------//
    CALL FILL_BLK
    {value_type := 'Bool', count_type := 'UInt'}
    (   IN                   := 0 ,
        COUNT                := 15 ,
        OUT                  := #tIL.Source[0]
    );


NETWORK
TITLE = Item 66 DV3113 interlock source : ON ZSC3107 Vessel inlet line Flowpath Indicator IN   ON ZSC3105 Vessel PW Supply Flowpath Indicator IN
    //------------------------------------------------------------------------//
    // Calculate the interlock condition:                                     //
    //------------------------------------------------------------------------//
    ON(;
    L "idbZSC2".f[16].p.read.mc.STATE;
    L "dbCONST".BLK.ZSC2.STATE.IN;
    ==I;
    );
ON(;
    L "idbZSC2".f[15].p.read.mc.STATE;
    L "dbCONST".BLK.ZSC2.STATE.IN;
    ==I;
    );
    = #tIL.Source[0];

NETWORK
TITLE = Item 66 DV3113 interlock source : A DV3115 Vessel PS Supply for PW Loop OPENED
    //------------------------------------------------------------------------//
    // Calculate the interlock condition:                                     //
    //------------------------------------------------------------------------//
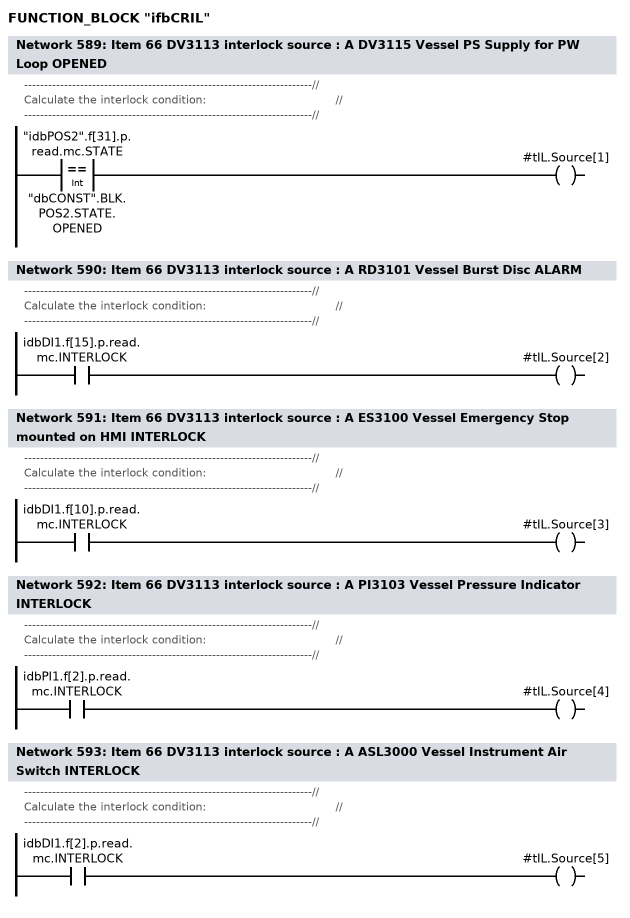
    A(;
    L "idbPOS2".f[31].p.read.mc.STATE;
    L "dbCONST".BLK.POS2.STATE.OPENED;
    ==I;
    );
    = #tIL.Source[1];

NETWORK
TITLE = Item 66 DV3113 interlock source : A RD3101 Vessel Burst Disc ALARM
    //------------------------------------------------------------------------//
    // Calculate the interlock condition:                                     //
    //------------------------------------------------------------------------//
    A idbDI1.f[15].p.read.mc.INTERLOCK;
    = #tIL.Source[2];

NETWORK
TITLE = Item 66 DV3113 interlock source : A ES3100 Vessel Emergency Stop mounted on HMI INTERLOCK
    //------------------------------------------------------------------------//
    // Calculate the interlock condition:                                     //
    //------------------------------------------------------------------------//
    A idbDI1.f[10].p.read.mc.INTERLOCK;
    = #tIL.Source[3];

NETWORK
TITLE = Item 66 DV3113 interlock source : A PI3103 Vessel Pressure Indicator INTERLOCK
    //------------------------------------------------------------------------//
    // Calculate the interlock condition:                                     //
    //------------------------------------------------------------------------//
    A idbPI1.f[2].p.read.mc.INTERLOCK;
    = #tIL.Source[4];

NETWORK
TITLE = Item 66 DV3113 interlock source : A ASL3000 Vessel Instrument Air Switch INTERLOCK
    //------------------------------------------------------------------------//
    // Calculate the interlock condition:                                     //
    //------------------------------------------------------------------------//
    A idbDI1.f[2].p.read.mc.INTERLOCK;
    = #tIL.Source[5];

NETWORK
TITLE = Item 66 DV3113 interlock source : AN ZSC3101 Vessel Manway Closed Indicator CLOSED
    //------------------------------------------------------------------------//
    // Calculate the interlock condition:                                     //
    //------------------------------------------------------------------------//
    AN(;
    L "idbZSC1".f[2].p.read.mc.STATE;
    L "dbCONST".BLK.ZSC1.STATE.CLOSED;
    ==I;
    );
    = #tIL.Source[6];


NETWORK
TITLE = Item 66 DV3113 : Number of interlocks
    //------------------------------------------------------------------------//
    // Number of interlocks
    //------------------------------------------------------------------------//
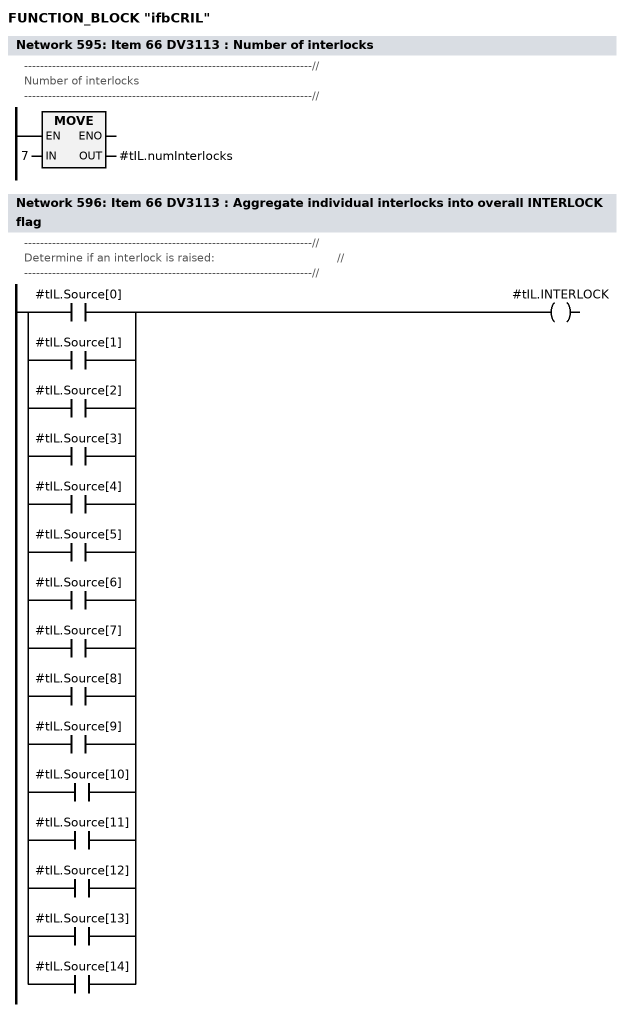
    L 7;
    T #tIL.numInterlocks;

NETWORK
TITLE = Item 66 DV3113 : Aggregate individual interlocks into overall INTERLOCK flag
    //------------------------------------------------------------------------//
    // Determine if an interlock is raised:                                   //
    //------------------------------------------------------------------------//
    O #tIL.Source[0];
    O #tIL.Source[1];
    O #tIL.Source[2];
    O #tIL.Source[3];
    O #tIL.Source[4];
    O #tIL.Source[5];
    O #tIL.Source[6];
    O #tIL.Source[7];
    O #tIL.Source[8];
    O #tIL.Source[9];
    O #tIL.Source[10];
    O #tIL.Source[11];
    O #tIL.Source[12];
    O #tIL.Source[13];
    O #tIL.Source[14];
    = #tIL.INTERLOCK;

NETWORK
TITLE = Item 66 DV3113 : Update the instance data
    //------------------------------------------------------------------------//
    // Update the instance DB with the calculated interlock flags:            //
    //------------------------------------------------------------------------//
    CALL MOVE
    {value_type := 'Variant'}
    (   IN                   := #tIL ,
        OUT                  := #p[66]
    );

NETWORK
TITLE = Item 67 DV3115 : PS Supply for PW Loop initialise variables
    //------------------------------------------------------------------------//
    // CRITICAL INTERLOCK   CRITICAL INTERLOCK   CRITICAL INTERLOCK   CRITICA //
    // CRITICAL INTERLOCK   CRITICAL INTERLOCK   CRITICAL INTERLOCK   CRITICA //
    //                                                                        //
    // Clear the interlock flag:                                              //
    //------------------------------------------------------------------------//
    A "alwaysLow";
    = #tIL.INTERLOCK;

    //------------------------------------------------------------------------//
    // Clear all interlock values to initialise them to off:                  //
    //------------------------------------------------------------------------//
    CALL FILL_BLK
    {value_type := 'Bool', count_type := 'UInt'}
    (   IN                   := 0 ,
        COUNT                := 15 ,
        OUT                  := #tIL.Source[0]
    );


NETWORK
TITLE = Item 67 DV3115 interlock source : ON ZSC3107 Vessel inlet line Flowpath Indicator IN   ON ZSC3105 Vessel PW Supply Flowpath Indicator IN
    //------------------------------------------------------------------------//
    // Calculate the interlock condition:                                     //
    //------------------------------------------------------------------------//
    ON(;
    L "idbZSC2".f[16].p.read.mc.STATE;
    L "dbCONST".BLK.ZSC2.STATE.IN;
    ==I;
    );
ON(;
    L "idbZSC2".f[15].p.read.mc.STATE;
    L "dbCONST".BLK.ZSC2.STATE.IN;
    ==I;
    );
    = #tIL.Source[0];

NETWORK
TITLE = Item 67 DV3115 interlock source : A DV3113 Vessel PW Supply Valve OPENED
    //------------------------------------------------------------------------//
    // Calculate the interlock condition:                                     //
    //------------------------------------------------------------------------//
